FUNCTION_BLOCK FB_UnitTestTarget01 EXTENDS FB_Target
VAR_INPUT
END_VAR
VAR_OUTPUT
END_VAR
VAR
	fbTestsuite:			FB_Testsuite;				// Testsuite
	sValue:					STRING;
END_VAR

SUPER^();

fbTestsuite();


CASE fbTestsuite.P_Testcase OF
	E_Testcase.Init:
		sValue:= 'Test';

	E_Testcase.Start:
		// First test case
		fbTestsuite.P_Assert.M_Equals_STRING('Test', sValue, 'Check string value "Test"');
		fbTestsuite.M_Testcase('FB_Target', T#1S, '', '', 1);
		
	// secound test case
	1:
		fbTestsuite.P_Assert.M_IsTRUE('Test2' <> sValue, 'Check string value "Test2"');
		fbTestsuite.M_Testcase('FB_Target', T#1S, '', '', E_Testcase.Done);
		
	E_Testcase.Done:
		
END_CASE

METHOD FB_init : BOOL
VAR_INPUT
	bInitRetains : BOOL; // if TRUE, the retain variables are initialized (warm start / cold start)
	bInCopyCode : BOOL;  // if TRUE, the instance afterwards gets moved into the copy code (online change)
END_VAR
//// Add Testsuite to Testsuites
fbTestsuites.M_Add(fbTestsuite);
fbTestsuite.P_File:= 'FB_Target';
END_METHOD

END_FUNCTION_BLOCK

(* stored: Version 1.1.0.1
   POU FB_UnitTestTarget01: Id {9b93d624-8032-0947-32f4-dcb0f3ba6bc3}, SpecialFunc None
   Method FB_init: Id {ae495c4e-2132-0530-24af-c77ded1a8942} *)
